FUNCTION_BLOCK GAIN
  (* Standard: 61499-2 *)
  (* Version 2013_12_10, Gabriel *)
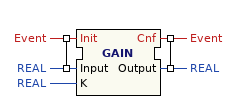
  EVENT_INPUT
    Init WITH Input;
  END_EVENT
  EVENT_OUTPUT
    Cnf WITH Output;
  END_EVENT
  VAR_INPUT
    Input : REAL;
    K : REAL;
  END_VAR
  VAR_OUTPUT
    Output : REAL;
  END_VAR
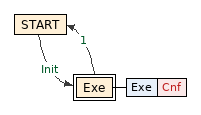
  EC_STATES
    Exe : Exe -> Cnf;
    START;
  END_STATES
  EC_TRANSITIONS
    START TO Exe := Init;
    Exe TO START := 1;
  END_TRANSITIONS
  ALGORITHM Exe IN Lua:
Output = K*Input
  END_ALGORITHM
END_FUNCTION_BLOCK
